FUNCTION_BLOCK FB_Test IMPLEMENTS I_Test
VAR_INPUT
END_VAR
VAR_OUTPUT
END_VAR
VAR
END_VAR

METHOD METH : BOOL
VAR_INPUT
END_VAR
END_METHOD

PROPERTY Name : STRING
GET
Name := 'Test';
END_GET
END_PROPERTY

END_FUNCTION_BLOCK

(* stored: Version 1.1.0.1, ProductVersion 3.1.4024.12
   POU FB_Test: Id {e29f903d-7e37-4dfb-b7bc-faafdeb7da7a}, SpecialFunc None
   Method METH: Id {9f908876-f844-416e-b279-14bd21525fed}
   Property Name: Id {a014e8f7-c5f0-4d75-be2e-cb82d3e30fd2}
   Get Get: Id {5ddd5ea9-6be2-4269-927b-8df3085c5ff5} *)
